SYSTEM SLIDERS (* FB_SLIDER Demo Configuration *)
  (* Standard: 61499-1 *)
  (* Version 0.1, 2006-02-02, JHC, Holobloc Inc., Saved to correct XML format. *)
  (* Version 0.0, 2004-09-04, JHC, Rockwell Automation *)
  APPLICATION APP1
  END_APPLICATION
  DEVICE DEV1 : FRAME_DEVICE(BOUNDS := [100,100,360,160])
    RESOURCE RES2 : PANEL_RESOURCE
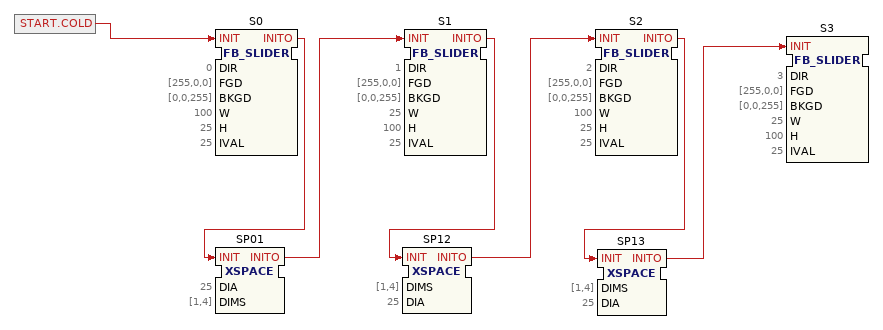
      FBS
        S0 : FB_SLIDER(DIR := 0, FGD := [255,0,0], BKGD := [0,0,255], W := 100, H := 25, IVAL := 25);
        S1 : FB_SLIDER(DIR := 1, FGD := [255,0,0], BKGD := [0,0,255], W := 25, H := 100, IVAL := 25);
        S2 : FB_SLIDER(DIR := 2, FGD := [255,0,0], BKGD := [0,0,255], W := 100, H := 25, IVAL := 25);
        S3 : FB_SLIDER(DIR := 3, FGD := [255,0,0], BKGD := [0,0,255], W := 25, H := 100, IVAL := 25);
        SP01 : XSPACE(DIA := 25, DIMS := [1,4]);
        SP12 : XSPACE(DIMS := [1,4], DIA := 25);
        SP13 : XSPACE(DIMS := [1,4], DIA := 25);
      END_FBS
      EVENT_CONNECTIONS
        START.COLD TO S0.INIT;
        S0.INITO TO SP01.INIT;
        SP01.INITO TO S1.INIT;
        S1.INITO TO SP12.INIT;
        SP12.INITO TO S2.INIT;
        S2.INITO TO SP13.INIT;
        SP13.INITO TO S3.INIT;
      END_CONNECTIONS
    END_RESOURCE
  END_DEVICE
END_SYSTEM
